TYPE "UDT_ZC_PINT"
VERSION : 0.1
   STRUCT
      Valor : Int;
      ValorAnterior : Int;
      Maximo : Int;   // Límite máximo
      Minimo : Int;   // Límite mínimo
   END_STRUCT;

END_TYPE

